{attribute 'qualified_only'}
{attribute 'strict'}
{attribute 'to_string'}
TYPE E_PuckLockerMode :
(
	Disabled := 0,
    Enabled := 1,
    EnabledWithEmptyPuckBypass := 2
);
END_TYPE

(* stored: Version 1.1.0.1, ProductVersion 3.1.4026.18
   DUT E_PuckLockerMode: Id {d9a0cb4d-94e8-441a-8e04-98c122b85541} *)
